(* IEC 61131-3 sources: PID-controller/sub blocks, 3 files *)

(* ---- DeadBand.st ---- *)
FUNCTION DeadBand : REAL
VAR_INPUT
	X        : REAL;
	deadZone : REAL;
END_VAR

(*
version 1.2	18. jan. 2011
programmer 	hugo
tested by		oscat

DEAD_BAND ist eine lineare Übertragungsfunktion mit Totzone. Die Funktion verschiebt den positiven Teil der Kurve um +L und den negativen Teil der Kurve um -L.
DEAD_BAND = X - L wenn X > L)
DEAD_BAND = X + L wenn X < -L
DEAD_BAND = 0 wenn Abs(X) <= L

*)

IF deadZone = 0.0 THEN
	DeadBand := X;
	RETURN;
END_IF
IF X > deadZone THEN
	DeadBand := X - deadZone;
ELSIF X < -deadZone THEN
	DeadBand := X + deadZone;
ELSE
	DeadBand := 0.0;
END_IF;

(* revision history
hm	2. nov. 2007	rev 1.0
	original version

hm	14. jun. 2008	rev 1.1
	improved performance

hm	18. jan. 2011	rev 1.2
	assign 0 before return
*)

(* ---- SCALE_R.st ---- *)
FUNCTION SCALE_R : REAL
VAR_INPUT
	X : REAL;
	I_LO : REAL;
	I_HI : REAL;
	O_LO : REAL;
	O_HI : REAL;
END_VAR

(*
version 1.2	11. jan. 2011
programmer 	hugo
tested by		oscat

Scale_R is used to translate and scale a REAL input x to a real output.
the input is limited to I_LO <= X <= I_HI.

*)

IF I_LO = I_HI THEN
	SCALE_R := O_LO;
ELSE
	SCALE_R := (O_HI - O_LO) / (I_HI - I_LO) * (LIMIT(I_LO, X, I_HI) - I_LO) + O_LO;
END_IF;

(* revision history
hm	18. may. 2008	rev 1.0
	original version

hm	13. nov. 2008	rev 1.1
	corrected formula for negative gradient

hm	11. jan 2011	rev 1.2
	avoid division by 0

*)

(* ---- LSim_PT1.st ---- *)
FUNCTION_BLOCK LSim_PT1
VAR_INPUT
    input     : REAL;      // input signal
    T         : REAL := 1.0;   // time constant T1 [sec]
    cycle     : REAL := 0.1;   // cyclic time [sec]
    bypass    : BOOL;      // resets all relevant parameters to ‘0’ including the output
END_VAR
VAR_OUTPUT
	error   : BOOL;   // error (tmLag1 <= 0)
    errorID : WORD;   // status (if tmLag1 <= 0 then status = 168001)
    out     : REAL;   // output signal (if error = FALSE)
END_VAR
VAR
	statRf1    : REAL;
    statRe1    : REAL;
    statOutput : REAL;
END_VAR
VAR CONSTANT
	ERR_BAD_FILTER_TIME : WORD := 16#8202;
	STATUS_NO_ERRORS    : WORD := 0;
END_VAR

{region BLOCK INFO HEADER}
 //===============================================================================
 // (company) / (c)Copyright (2024)
 //-------------------------------------------------------------------------------
 // Title:            PT1
 // Comment/Function: First order filter (low-pass)
 // Library/Family:   LSim
 // Author:           controltheplant
 // Tested with:      Codesys Control Win V3
 // Engineering:      Codesys 64 V3.5.19
 // Restrictions:     cyclic interrupt
 // Requirements:     (hardware, technological package, memory needed, etc.)
 //-------------------------------------------------------------------------------
 // Change log table:
 // Version  | Date       | Expert in charge       | Changes applied
 //----------|------------|------------------------|------------------------------
 // 01.00.00 | 2023-09-18 |                        | First released version
 //===============================================================================
{endregion}

{region DESCRIPTION}
(*
FB “LSim_PT1” simulates a PT1 element. The PT1 element is a proportional transfer element with first-order order delay.
              gain
  F(s) = ---------------
          tmLag1 * s + 1
*)
{endregion}

IF T < 0 THEN
    error := TRUE;
    errorID := ERR_BAD_FILTER_TIME; // Parameter Error
    statOutput := 0;
    out := 0;
    RETURN;
ELSIF T = 0.0 THEN
	statOutput := input;
	out := statOutput;
	RETURN;
ELSE
    error := FALSE;
    errorID := STATUS_NO_ERRORS; // no error
END_IF;

IF bypass THEN
    statOutput := input;
	RETURN;
END_IF;

// possible improvement: calculate exp only when parameter T changes
// Z-parameters For Laplace PT1-System
statRe1 := - EXP(-cycle/T);
statRf1 := 1 + statRe1;

// Differencial Equation of PT1-System
statOutput := input*statRf1 - statOutput*statRe1;

out := statOutput;
